// EL2032 | 2-channel digital output terminal 24 V DC, 2 A
FUNCTION_BLOCK EL2032

VAR_INPUT
    En: BOOL;
    iTerminal_ID : INT;
    ErrorSystem : POINTER TO ST_ErrorSystem;
END_VAR

VAR_OUTPUT
    EnO: BOOL;
    bError: BOOL;
	sErrorMessage       : STRING;
END_VAR

VAR
    WcState_WcState AT %I* : BOOL := FALSE;
    InfoData_State  AT %I* : UINT := 0;

    //FB-s
    EL2032_Error    : FB_TerminalError;
END_VAR

(*
* TODO: Test on hardware
*)

EnO:=En;

EL2032_Error(
    En := TRUE,
    iTerminal_ID := iTerminal_ID,
    bWcState := FALSE,
    uiInfoData_State := InfoData_State,
    pErrorSystem := ErrorSystem,
    bError => bError,
);

IF bError THEN
	sErrorMessage:=EL2032_Error.ErrorData.sErrorMessage;
ELSE
	sErrorMessage:='';
END_IF

END_FUNCTION_BLOCK

(* stored: Version 1.1.0.1, ProductVersion 3.1.4024.0
   POU EL2032: Id {86656376-936d-43d8-a7e4-bd6e7e703ffd}, SpecialFunc None *)
